// TIA Portal V16 program export: 1 tag tables, 0 data types, 0 data blocks, 2 code blocks (in call order from the OBs), 1 instance data blocks

VAR_GLOBAL   // PLC tag table "Table de variables standard"
   Bascule AT %M0.0 : Bool;
   Bit1 AT %M0.1 : Bool;
   Bit2 AT %M0.2 : Bool;
   Bit3 AT %M0.3 : Bool;
   Sensor1 AT %M0.4 : Bool;
   Sensor2 AT %M0.5 : Bool;
   Coil20 AT %M0.6 : Bool;
END_VAR

ORGANIZATION_BLOCK "Main"   // OB1, LAD, ProgramCycle
TITLE = "Main Program Sweep (Cycle)"
{ S7_Optimized_Access := 'TRUE' }
VERSION : 0.1
// stored: AutoNumber true, IsIECCheckEnabled false, SetENOAutomatically false
BEGIN

REGION Network 1
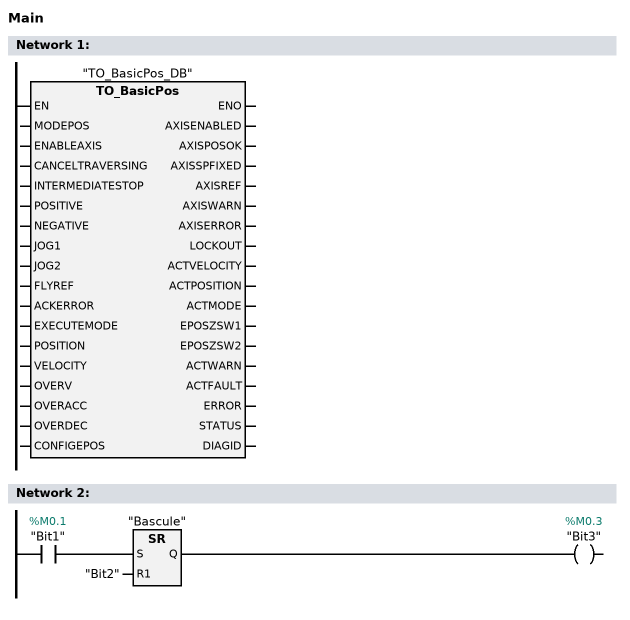
   RUNG wire#powerrail
      "TO_BasicPos_DB".TO_BasicPos(ModePos :=, EnableAxis :=, CancelTraversing :=, IntermediateStop :=, Positive :=, Negative :=, Jog1 :=, Jog2 :=, FlyRef :=, AckError :=, ExecuteMode :=, Position :=, Velocity :=, OverV :=, OverAcc :=, OverDec :=, ConfigEPos :=, AxisEnabled =>, AxisPosOk =>, AxisSpFixed =>, AxisRef =>, AxisWarn =>, AxisError =>, Lockout =>, ActVelocity =>, ActPosition =>, ActMode =>, EPosZSW1 =>, EPosZSW2 =>, ActWarn =>, ActFault =>, Error =>, Status =>, DiagId =>)
   END_RUNG
   // the same network as SCL:
   "TO_BasicPos_DB"();   // TO_BasicPos
END_REGION

REGION Network 2
   RUNG wire#powerrail
      Contact( "Bit1" )
      S_SR(operand := "Bascule", r1 := "Bit2")
      Coil( "Bit3" )
   END_RUNG
   // the same network as SCL:
   IF "Bit1" THEN
       "Bascule" := TRUE;   // SR flip-flop
   END_IF;
   IF "Bit2" THEN "Bascule" := FALSE; END_IF;
   "Bit3" := "Bascule";
END_REGION
END_ORGANIZATION_BLOCK

FUNCTION_BLOCK "Analog scaling output"
{ S7_Optimized_Access := 'TRUE' }
VERSION : 0.1
   VAR_INPUT 
      In1 : Bool;
      In2 : Bool;
   END_VAR

   VAR_OUTPUT 
      Out20 : Bool;
   END_VAR


BEGIN
	IF #In1 AND NOT #In2 THEN
	    // Statement section IF
	    #Out20 := true;
	END_IF;
	
END_FUNCTION_BLOCK

DATA_BLOCK "Analog scaling output_DB"   // DB3
VERSION : 0.1
// stored: AutoNumber true, InstanceOfName Analog scaling output, InstanceOfType FB
"Analog scaling output"
BEGIN
END_DATA_BLOCK
